// TIA Portal V16 export
// export: Created 2022-09-01T13:36:46.8108244Z, ExportSetting WithDefaults, DisplayName Totally Integrated Automation Portal, DisplayVersion V16, DisplayName TIA Portal Version Control Interface, DisplayVersion V16, DisplayName TIA Portal Openness, DisplayVersion V16, DisplayName STEP 7 Professional, DisplayVersion V16, DisplayName STEP 7 Safety, DisplayVersion V16, DisplayName WinCC Advanced, DisplayVersion V16
FUNCTION "Proc_Analog_FQ301" : Void   // FC12, LAD
{ S7_Optimized_Access := 'TRUE' }
VERSION : 0.1
// stored: AutoNumber true, IsIECCheckEnabled false, SetENOAutomatically false, UDAEnableTagReadback false
   VAR_INPUT
      Analog_Input_Value : Int;
   END_VAR
   VAR_OUTPUT
      "Caudal_em_m3/h" : Real;
   END_VAR
   VAR_TEMP
      "Caudal_em_%" : Real;
   END_VAR
BEGIN

REGION Network 1
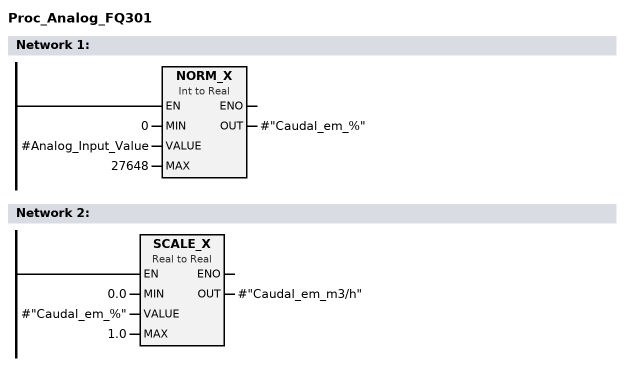
   RUNG wire#powerrail
      { S7_Templates := "[SrcType := Int, DestType := Real]"; S7_GenerateENO := "TRUE" } Normalize(min := 0, value := #Analog_Input_Value, max := 27648, out => #"Caudal_em_%")
   END_RUNG
   // the same network as SCL:
   #"Caudal_em_%" := NORM_X(MIN := 0, VALUE := #Analog_Input_Value, MAX := 27648);
END_REGION

REGION Network 2
   RUNG wire#powerrail
      { S7_Templates := "[SrcType := Real, DestType := Real]"; S7_GenerateENO := "TRUE" } Scale(min := 0.0, value := #"Caudal_em_%", max := 1.0, out => #"Caudal_em_m3/h")
   END_RUNG
   // the same network as SCL:
   #"Caudal_em_m3/h" := SCALE_X(MIN := 0.0, VALUE := #"Caudal_em_%", MAX := 1.0);
END_REGION
END_FUNCTION
